(* Logix 5000 project; controller cow Emulate 5570 rev 36.11; software revision 36.00; part 2 of 6 *)

ADD_ON_INSTRUCTION RTOS_Format   (* revision 1.0 *)
VAR_INPUT
   Source : REAL; {required}
END_VAR
VAR_IN_OUT
   Dest : String20; {required}
END_VAR
VAR
   DotS : STRING := '.'; {access None}
   dotPos : DINT[2]; {access None}
   dotPos_1 : DINT; {access None}
   Blank : STRING := ' '; {access None}
END_VAR

ROUTINE Logic   (* ladder *)
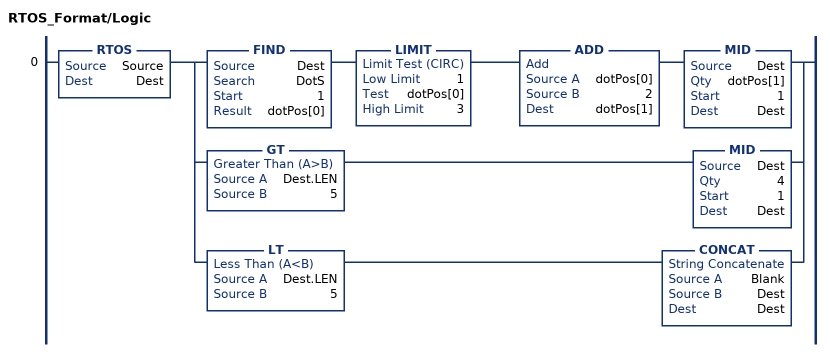
   0: RTOS(Source,Dest)[FIND(Dest,DotS,1,dotPos[0]) LIMIT(1,dotPos[0],3) ADD(dotPos[0],2,dotPos[1]) MID(Dest,dotPos[1],1,Dest) ,GT(Dest.LEN,5) MID(Dest,4,1,Dest) ,LT(Dest.LEN,5) CONCAT(Blank,Dest,Dest) ];
END_ROUTINE
END_ADD_ON_INSTRUCTION

ADD_ON_INSTRUCTION SCALE_WEIGHT   (* revision 1.0 *)
VAR_INPUT
   BCD0 : ALIAS FOR BCD.0; {access None, visible}
   BCD1 : ALIAS FOR BCD.1; {access None, visible}
   BCD2 : ALIAS FOR BCD.2; {access None, visible}
   BCD3 : ALIAS FOR BCD.3; {access None, visible}
   BCD4 : ALIAS FOR BCD.4; {access None, visible}
   BCD5 : ALIAS FOR BCD.5; {access None, visible}
   BCD6 : ALIAS FOR BCD.6; {access None, visible}
   BCD7 : ALIAS FOR BCD.7; {access None, visible}
   BCD8 : ALIAS FOR BCD.8; {access None, visible}
   BCD9 : ALIAS FOR BCD.9; {access None, visible}
   BCD10 : ALIAS FOR BCD.10; {access None, visible}
   BCD11 : ALIAS FOR BCD.11; {access None, visible}
   BCD12 : ALIAS FOR BCD.12; {access None, visible}
   BCD13 : ALIAS FOR BCD.13; {access None, visible}
   BCD14 : ALIAS FOR BCD.14; {access None, visible}
   BCD15 : ALIAS FOR BCD.15; {access None, visible}
END_VAR
VAR_OUTPUT
   DM : BOOL; {access Read Only, visible}
   DMGL : BOOL; {access Read Only, visible}
END_VAR
VAR_INPUT
   PB : BOOL; {visible}
END_VAR
VAR_OUTPUT
   SV : BOOL; {access Read Only, visible}
END_VAR
VAR_INPUT
   LL : BOOL; {visible}
END_VAR
VAR_OUTPUT
   PB2 : BOOL;
   DM2 : BOOL;
END_VAR
VAR_INPUT
   Sign : BOOL;
END_VAR
VAR_OUTPUT
   Value : INT; {access Read Only, visible}
END_VAR
VAR_IN_OUT
   Sys : Sys_Data; {required}
END_VAR
VAR
   BCD : INT; {access None}
END_VAR

ROUTINE Logic   (* ladder *)
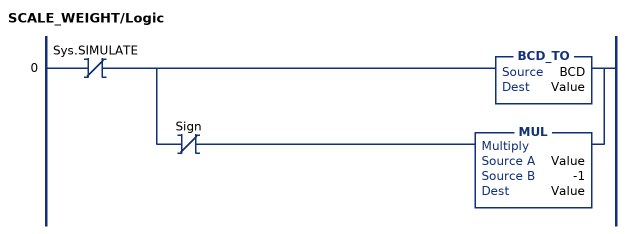
   0: XIO(Sys.SIMULATE)[BCD_TO(BCD,Value) ,XIO(Sign) MUL(Value,-1,Value) ];
END_ROUTINE
END_ADD_ON_INSTRUCTION

ADD_ON_INSTRUCTION Speed_RPM   (* revision 1.0 *)
VAR_IN_OUT
   Motor : MotorX; {required}
END_VAR
VAR_INPUT
   RPM_Low : INT := 60; {visible}
END_VAR
VAR_OUTPUT
   RPM : INT; {visible}
END_VAR
VAR
   Timer : TIMER := (PRE := 5000); {access None}
   temp : INT[10]; {access None}
   Sort_control : CONTROL := (LEN := 10); {access None}
   RPM_AVG : REAL; {access None}
   rpm_ons : DINT; {access None}
   No_Input : BOOL; {access None}
   FIFO_control : CONTROL := (LEN := 10, POS := 10); {access None}
   FIFO : INT[11]; {access None}
   AVE_Control : CONTROL := (LEN := 8); {access None}
   Motor_Start : TIMER := (PRE := 5000); {access None}
   Delay : TIMER := (PRE := 5000); {access None}
   RUNTIME : TIMER := (PRE := 14400000, ACC := 14400000); {access None}
END_VAR

ROUTINE Logic   (* ladder *)
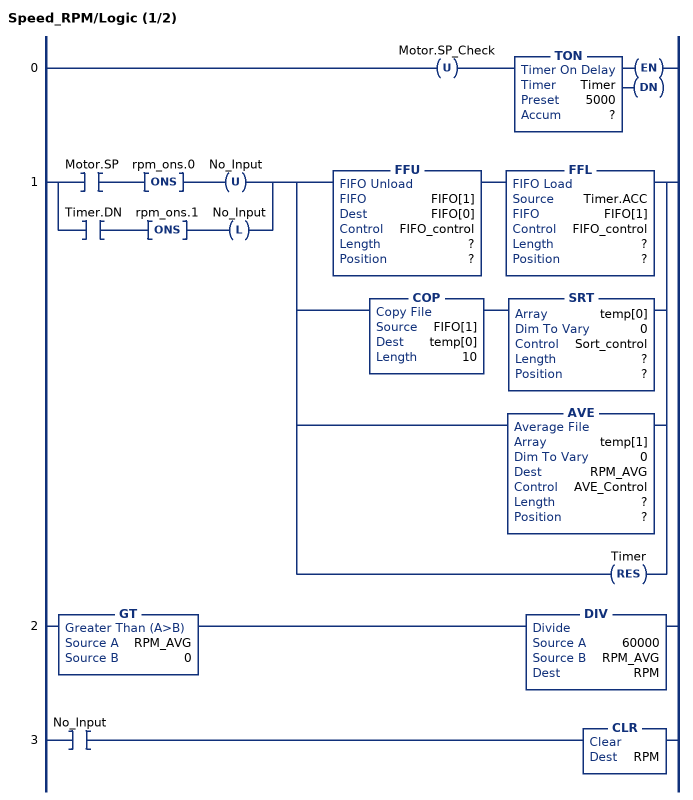
   0: OTU(Motor.SP_Check)TON(Timer,?,?);
   1: [XIC(Motor.SP) ONS(rpm_ons.0) OTU(No_Input) ,XIC(Timer.DN) ONS(rpm_ons.1) OTL(No_Input) ][FFU(FIFO[1],FIFO[0],FIFO_control,?,?) FFL(Timer.ACC,FIFO[1],FIFO_control,?,?) ,COP(FIFO[1],temp[0],10) SRT(temp[0],0,Sort_control,?,?) ,AVE(temp[1],0,RPM_AVG,AVE_Control,?,?) ,RES(Timer) ];
   2: GT(RPM_AVG,0)DIV(60000,RPM_AVG,RPM);
   3: XIC(No_Input)CLR(RPM);
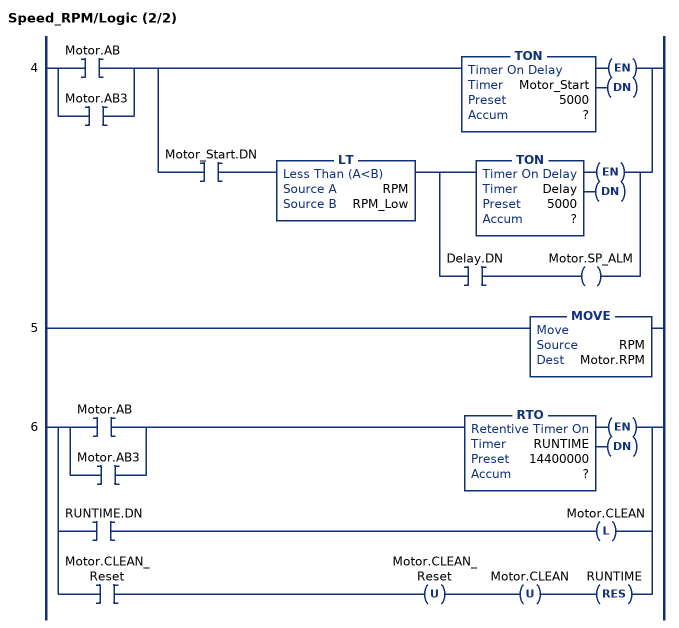
   4: [XIC(Motor.AB) ,XIC(Motor.AB3) ][TON(Motor_Start,?,?) ,XIC(Motor_Start.DN) LT(RPM,RPM_Low) [TON(Delay,?,?) ,XIC(Delay.DN) OTE(Motor.SP_ALM) ] ];
   5: MOVE(RPM,Motor.RPM);
   6: [[XIC(Motor.AB) ,XIC(Motor.AB3) ] RTO(RUNTIME,?,?) ,XIC(RUNTIME.DN) OTL(Motor.CLEAN) ,XIC(Motor.CLEAN_Reset) OTU(Motor.CLEAN_Reset) OTU(Motor.CLEAN) RES(RUNTIME) ];
END_ROUTINE
END_ADD_ON_INSTRUCTION

ADD_ON_INSTRUCTION Str_Len_Fix   (* revision 1.0 *)
VAR_IN_OUT
   Str : STRING; {required}
END_VAR
VAR_INPUT
   Len : DINT; {required}
END_VAR

ROUTINE Logic   (* ladder *)
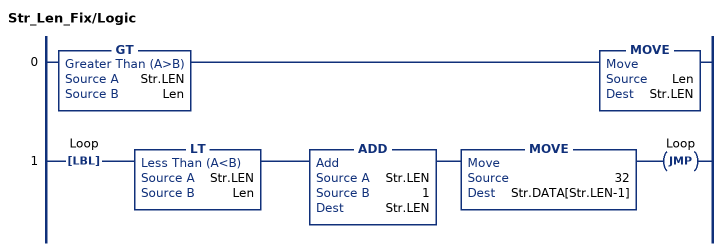
   0: GT(Str.LEN,Len)MOVE(Len,Str.LEN);
   1: LBL(Loop)LT(Str.LEN,Len)ADD(Str.LEN,1,Str.LEN)MOVE(32,Str.DATA[Str.LEN-1])JMP(Loop);
END_ROUTINE
END_ADD_ON_INSTRUCTION

ADD_ON_INSTRUCTION System_Data   (* revision 1.0 *)
VAR_OUTPUT
   MC : BOOL; {visible}
END_VAR
VAR_IN_OUT
   SYS : Sys_Data; {required}
   STS : INT; {required}
   sys_common : System_Common; {required}
END_VAR
VAR
   ons : DINT; {access None}
   EM_TIMER : TIMER := (PRE := 5000); {access None}
   BIN_SEL_PRE : DINT; {access None}
   BIN_SELS_PRE : DINT; {access None}
   Report_Log : TIMER := (PRE := 5000); {access None}
   Err_Reset_Timer : TIMER := (PRE := 1000); {access None}
END_VAR

ROUTINE Logic   (* ladder *)
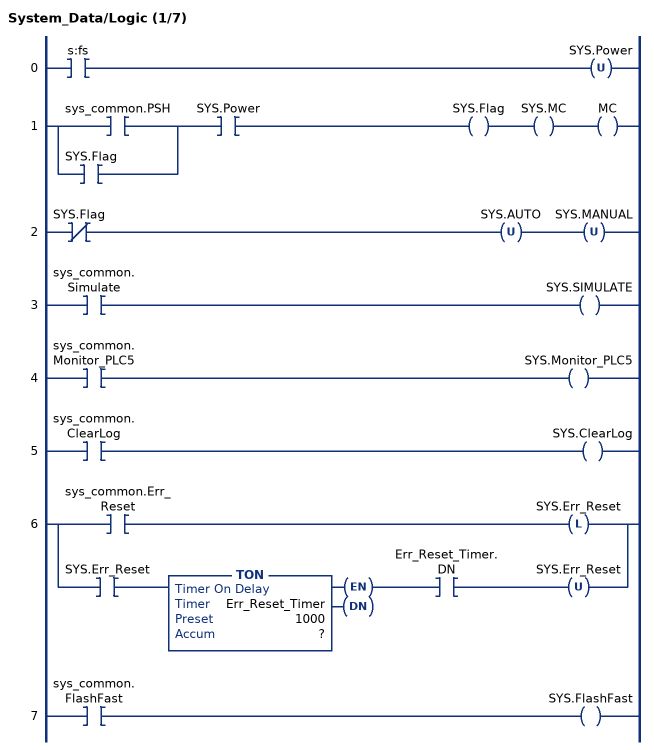
   0: XIC(s:fs)OTU(SYS.Power);
   1: [XIC(sys_common.PSH) ,XIC(SYS.Flag) ]XIC(SYS.Power)OTE(SYS.Flag)OTE(SYS.MC)OTE(MC);
   2: XIO(SYS.Flag)OTU(SYS.AUTO)OTU(SYS.MANUAL);
   3: XIC(sys_common.Simulate)OTE(SYS.SIMULATE);
   4: XIC(sys_common.Monitor_PLC5)OTE(SYS.Monitor_PLC5);
   5: XIC(sys_common.ClearLog)OTE(SYS.ClearLog);
   6: [XIC(sys_common.Err_Reset) OTL(SYS.Err_Reset) ,XIC(SYS.Err_Reset) TON(Err_Reset_Timer,?,?) XIC(Err_Reset_Timer.DN) OTU(SYS.Err_Reset) ];
   7: XIC(sys_common.FlashFast)OTE(SYS.FlashFast);
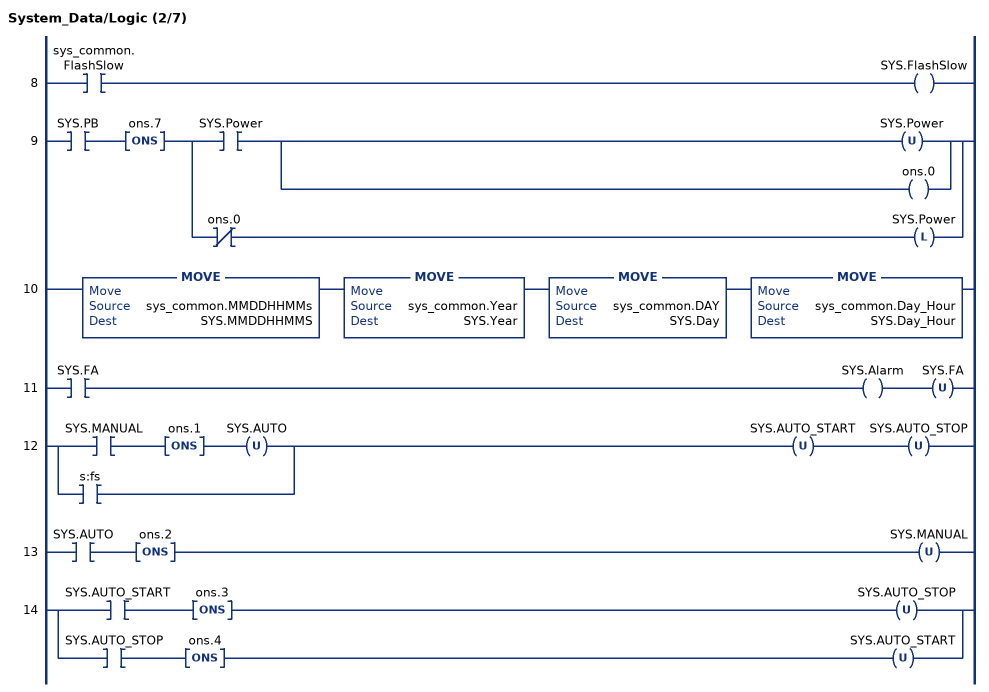
   8: XIC(sys_common.FlashSlow)OTE(SYS.FlashSlow);
   9: XIC(SYS.PB)ONS(ons.7)[XIC(SYS.Power) [OTU(SYS.Power) ,OTE(ons.0) ] ,XIO(ons.0) OTL(SYS.Power) ];
   10: MOVE(sys_common.MMDDHHMMs,SYS.MMDDHHMMS)MOVE(sys_common.Year,SYS.Year)MOVE(sys_common.DAY,SYS.Day)MOVE(sys_common.Day_Hour,SYS.Day_Hour);
   11: XIC(SYS.FA)OTE(SYS.Alarm)OTU(SYS.FA);
   12: [XIC(SYS.MANUAL) ONS(ons.1) OTU(SYS.AUTO) ,XIC(s:fs) ]OTU(SYS.AUTO_START)OTU(SYS.AUTO_STOP);
   13: XIC(SYS.AUTO)ONS(ons.2)OTU(SYS.MANUAL);
   14: [XIC(SYS.AUTO_START) ONS(ons.3) OTU(SYS.AUTO_STOP) ,XIC(SYS.AUTO_STOP) ONS(ons.4) OTU(SYS.AUTO_START) ];
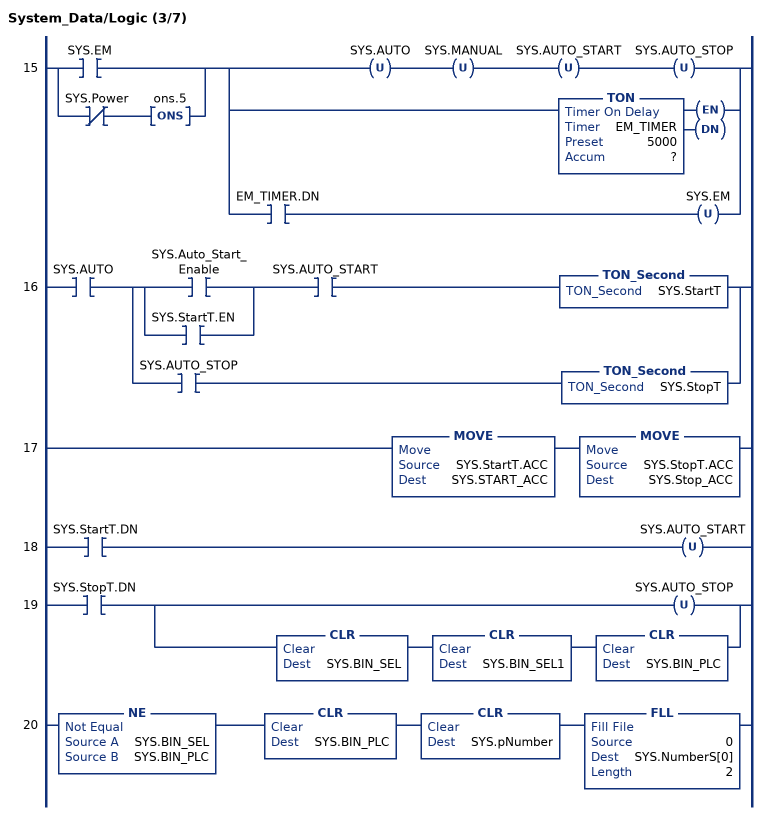
   15: [XIC(SYS.EM) ,XIO(SYS.Power) ONS(ons.5) ][OTU(SYS.AUTO) OTU(SYS.MANUAL) OTU(SYS.AUTO_START) OTU(SYS.AUTO_STOP) ,TON(EM_TIMER,?,?) ,XIC(EM_TIMER.DN) OTU(SYS.EM) ];
   16: XIC(SYS.AUTO)[[XIC(SYS.Auto_Start_Enable) ,XIC(SYS.StartT.EN) ] XIC(SYS.AUTO_START) TON_Second(SYS.StartT) ,XIC(SYS.AUTO_STOP) TON_Second(SYS.StopT) ];
   17: MOVE(SYS.StartT.ACC,SYS.START_ACC)MOVE(SYS.StopT.ACC,SYS.Stop_ACC);
   18: XIC(SYS.StartT.DN)OTU(SYS.AUTO_START);
   19: XIC(SYS.StopT.DN)[OTU(SYS.AUTO_STOP) ,CLR(SYS.BIN_SEL) CLR(SYS.BIN_SEL1) CLR(SYS.BIN_PLC) ];
   20: NE(SYS.BIN_SEL,SYS.BIN_PLC)CLR(SYS.BIN_PLC)CLR(SYS.pNumber)FLL(0,SYS.NumberS[0],2);
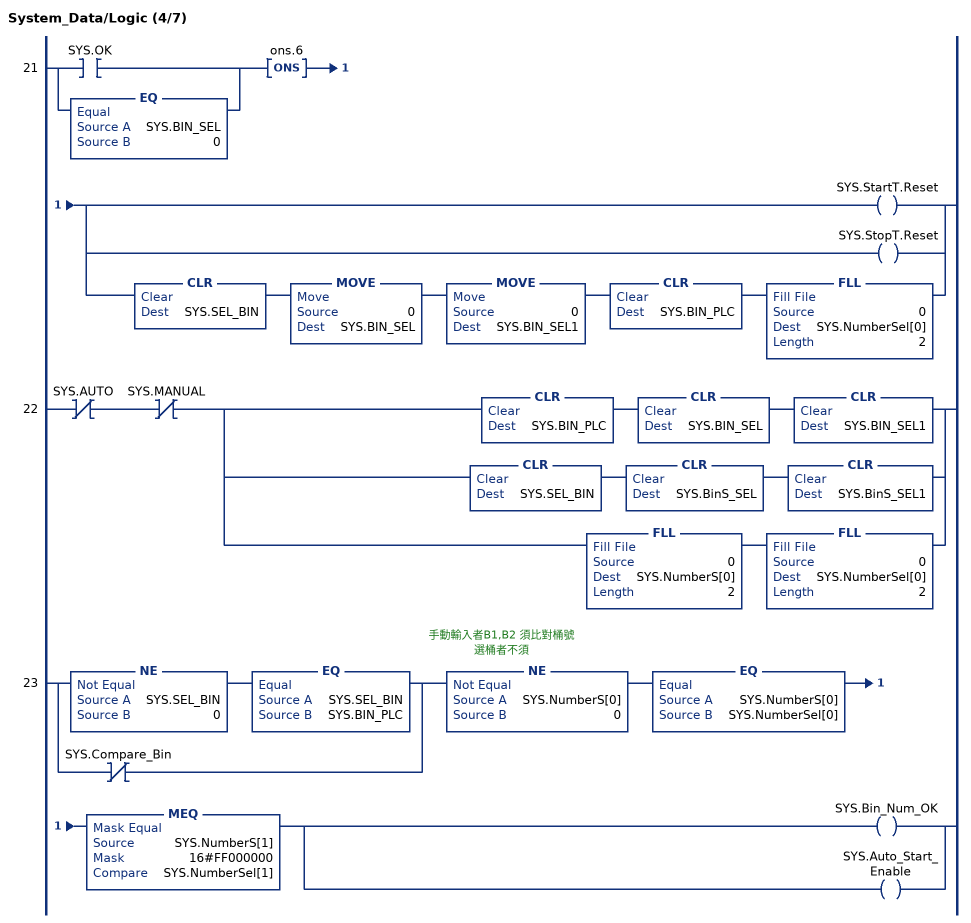
   21: [XIC(SYS.OK) ,EQ(SYS.BIN_SEL,0) ]ONS(ons.6)[OTE(SYS.StartT.Reset) ,OTE(SYS.StopT.Reset) ,CLR(SYS.SEL_BIN) MOVE(0,SYS.BIN_SEL) MOVE(0,SYS.BIN_SEL1) CLR(SYS.BIN_PLC) FLL(0,SYS.NumberSel[0],2) ];
   22: XIO(SYS.AUTO)XIO(SYS.MANUAL)[CLR(SYS.BIN_PLC) CLR(SYS.BIN_SEL) CLR(SYS.BIN_SEL1) ,CLR(SYS.SEL_BIN) CLR(SYS.BinS_SEL) CLR(SYS.BinS_SEL1) ,FLL(0,SYS.NumberS[0],2) FLL(0,SYS.NumberSel[0],2) ];
   // 手動輸入者B1,B2 須比對桶號
   // 選桶者不須
   23: [NE(SYS.SEL_BIN,0) EQ(SYS.SEL_BIN,SYS.BIN_PLC) ,XIO(SYS.Compare_Bin) ]NE(SYS.NumberS[0],0)EQ(SYS.NumberS[0],SYS.NumberSel[0])MEQ(SYS.NumberS[1],16#FF000000,SYS.NumberSel[1])[OTE(SYS.Bin_Num_OK) ,OTE(SYS.Auto_Start_Enable) ];
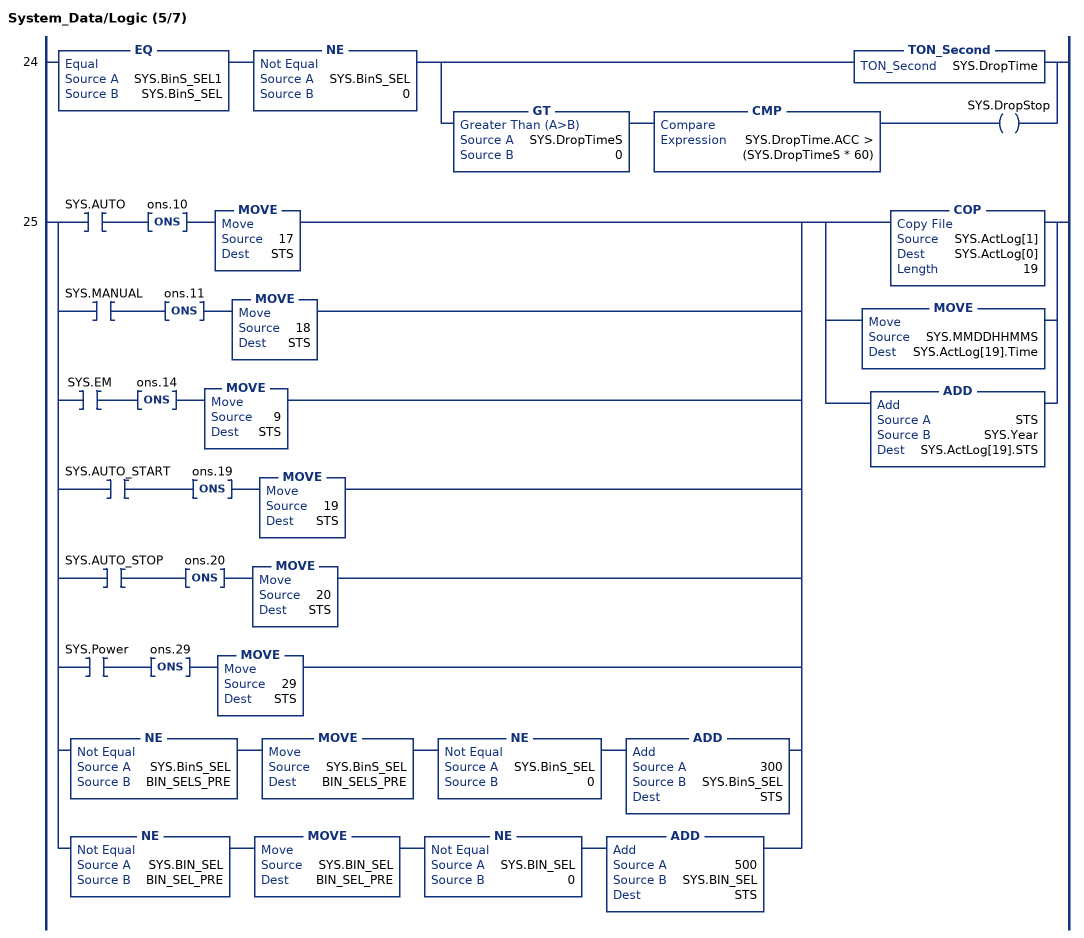
   24: EQ(SYS.BinS_SEL1,SYS.BinS_SEL)NE(SYS.BinS_SEL,0)[TON_Second(SYS.DropTime) ,GT(SYS.DropTimeS,0) CMP(SYS.DropTime.ACC > (SYS.DropTimeS * 60)) OTE(SYS.DropStop) ];
   25: [XIC(SYS.AUTO) ONS(ons.10) MOVE(17,STS) ,XIC(SYS.MANUAL) ONS(ons.11) MOVE(18,STS) ,XIC(SYS.EM) ONS(ons.14) MOVE(9,STS) ,XIC(SYS.AUTO_START) ONS(ons.19) MOVE(19,STS) ,XIC(SYS.AUTO_STOP) ONS(ons.20) MOVE(20,STS) ,XIC(SYS.Power) ONS(ons.29) MOVE(29,STS) ,NE(SYS.BinS_SEL,BIN_SELS_PRE) MOVE(SYS.BinS_SEL,BIN_SELS_PRE) NE(SYS.BinS_SEL,0) ADD(300,SYS.BinS_SEL,STS) ,NE(SYS.BIN_SEL,BIN_SEL_PRE) MOVE(SYS.BIN_SEL,BIN_SEL_PRE) NE(SYS.BIN_SEL,0) ADD(500,SYS.BIN_SEL,STS) ][COP(SYS.ActLog[1],SYS.ActLog[0],19) ,MOVE(SYS.MMDDHHMMS,SYS.ActLog[19].Time) ,ADD(STS,SYS.Year,SYS.ActLog[19].STS) ];
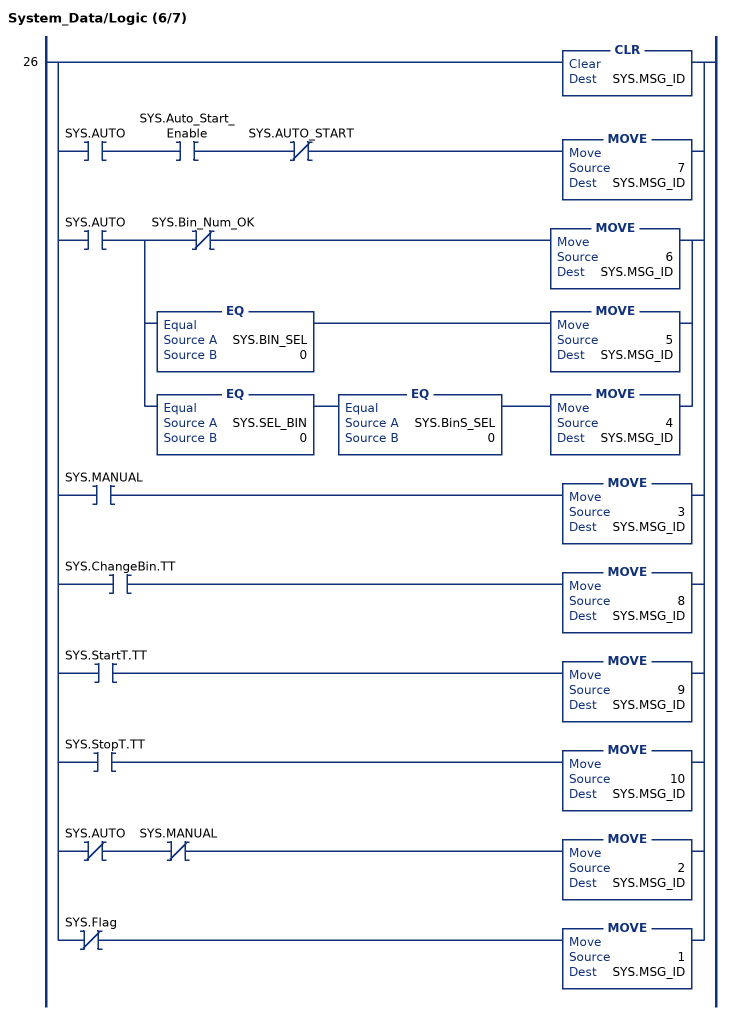
   26: [CLR(SYS.MSG_ID) ,XIC(SYS.AUTO) XIC(SYS.Auto_Start_Enable) XIO(SYS.AUTO_START) MOVE(7,SYS.MSG_ID) ,XIC(SYS.AUTO) [XIO(SYS.Bin_Num_OK) MOVE(6,SYS.MSG_ID) ,EQ(SYS.BIN_SEL,0) MOVE(5,SYS.MSG_ID) ,EQ(SYS.SEL_BIN,0) EQ(SYS.BinS_SEL,0) MOVE(4,SYS.MSG_ID) ] ,XIC(SYS.MANUAL) MOVE(3,SYS.MSG_ID) ,XIC(SYS.ChangeBin.TT) MOVE(8,SYS.MSG_ID) ,XIC(SYS.StartT.TT) MOVE(9,SYS.MSG_ID) ,XIC(SYS.StopT.TT) MOVE(10,SYS.MSG_ID) ,XIO(SYS.AUTO) XIO(SYS.MANUAL) MOVE(2,SYS.MSG_ID) ,XIO(SYS.Flag) MOVE(1,SYS.MSG_ID) ];
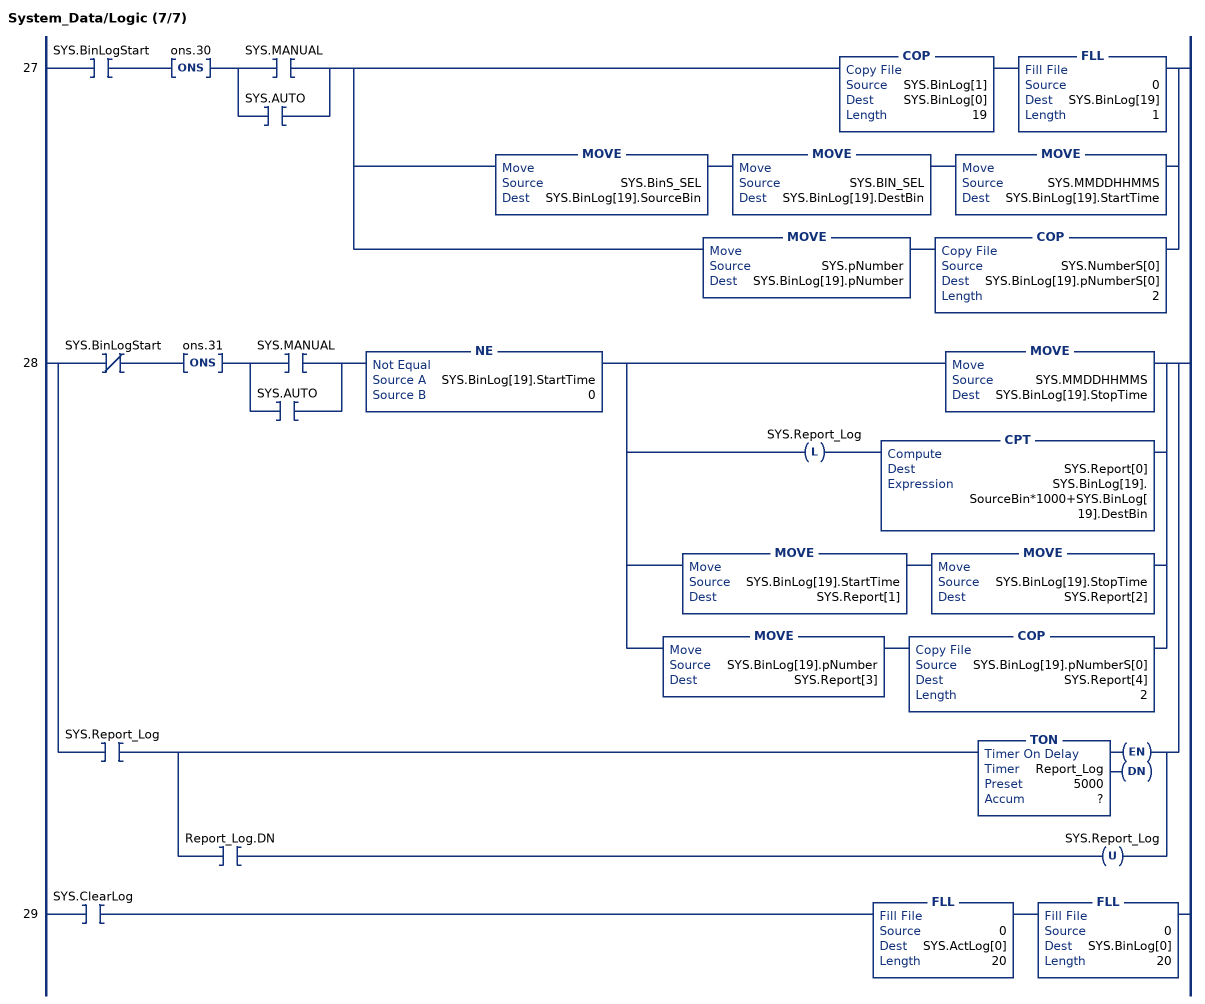
   27: XIC(SYS.BinLogStart)ONS(ons.30)[XIC(SYS.MANUAL) ,XIC(SYS.AUTO) ][COP(SYS.BinLog[1],SYS.BinLog[0],19) FLL(0,SYS.BinLog[19],1) ,MOVE(SYS.BinS_SEL,SYS.BinLog[19].SourceBin) MOVE(SYS.BIN_SEL,SYS.BinLog[19].DestBin) MOVE(SYS.MMDDHHMMS,SYS.BinLog[19].StartTime) ,MOVE(SYS.pNumber,SYS.BinLog[19].pNumber) COP(SYS.NumberS[0],SYS.BinLog[19].pNumberS[0],2) ];
   28: [XIO(SYS.BinLogStart) ONS(ons.31) [XIC(SYS.MANUAL) ,XIC(SYS.AUTO) ] NE(SYS.BinLog[19].StartTime,0) [MOVE(SYS.MMDDHHMMS,SYS.BinLog[19].StopTime) ,OTL(SYS.Report_Log) CPT(SYS.Report[0],SYS.BinLog[19].SourceBin*1000+SYS.BinLog[19].DestBin) ,MOVE(SYS.BinLog[19].StartTime,SYS.Report[1]) MOVE(SYS.BinLog[19].StopTime,SYS.Report[2]) ,MOVE(SYS.BinLog[19].pNumber,SYS.Report[3]) COP(SYS.BinLog[19].pNumberS[0],SYS.Report[4],2) ] ,XIC(SYS.Report_Log) [TON(Report_Log,?,?) ,XIC(Report_Log.DN) OTU(SYS.Report_Log) ] ];
   29: XIC(SYS.ClearLog)FLL(0,SYS.ActLog[0],20)FLL(0,SYS.BinLog[0],20);
END_ROUTINE
END_ADD_ON_INSTRUCTION

ADD_ON_INSTRUCTION TON_Second   (* revision 1.0, ExecuteEnableInFalse *)
VAR_OUTPUT
   EN : ALIAS FOR Timer.EN; {access None, visible}
   DN : ALIAS FOR Timer.DN; {access None, visible}
   TT : ALIAS FOR Timer.TT; {access None, visible}
   Reset : BOOL;
END_VAR
VAR_INPUT
   PRE : DINT; {visible}
END_VAR
VAR_OUTPUT
   ACC : DINT; {visible}
END_VAR
VAR
   Timer : TIMER; {access None}
   ACC_Temp : DINT; {access None}
END_VAR

ROUTINE EnableInFalse   (* ladder *)
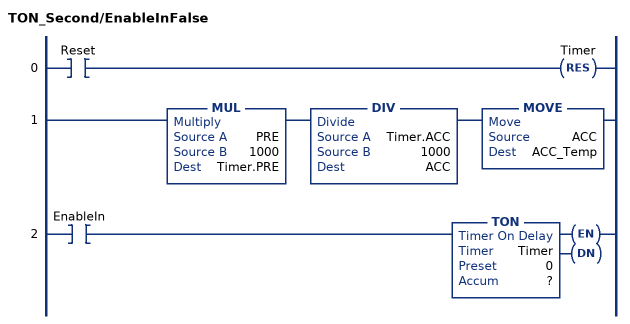
   0: XIC(Reset)RES(Timer);
   1: MUL(PRE,1000,Timer.PRE)DIV(Timer.ACC,1000,ACC)MOVE(ACC,ACC_Temp);
   2: XIC(EnableIn)TON(Timer,?,?);
END_ROUTINE

ROUTINE Logic   (* ladder *)
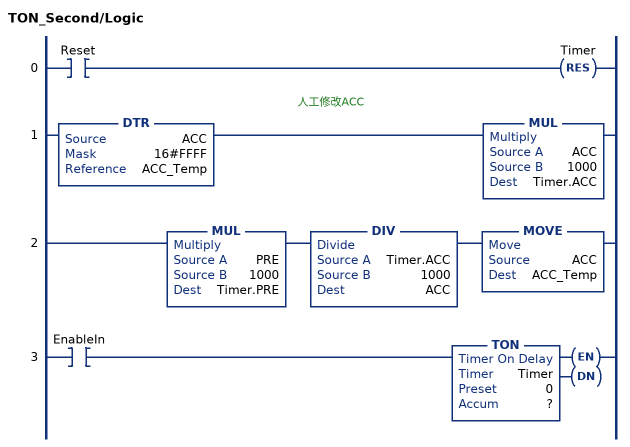
   0: XIC(Reset)RES(Timer);
   // 人工修改ACC
   1: DTR(ACC,16#FFFF,ACC_Temp)MUL(ACC,1000,Timer.ACC);
   2: MUL(PRE,1000,Timer.PRE)DIV(Timer.ACC,1000,ACC)MOVE(ACC,ACC_Temp);
   3: XIC(EnableIn)TON(Timer,?,?);
END_ROUTINE
END_ADD_ON_INSTRUCTION

ADD_ON_INSTRUCTION Valve   (* revision 1.0 *)
VAR_INPUT
   LSO : BOOL; {visible}
   LSK : BOOL; {visible}
END_VAR
VAR_OUTPUT
   SV : BOOL; {visible}
   Auto_On : BOOL;
   Manual_On : BOOL;
   Manual : BOOL; {visible}
   FA : BOOL; {visible}
   OPEN : BOOL; {visible}
   InterLock : BOOL; {access Read Only, visible}
   Auto : BOOL;
   PB : BOOL;
   GL : BOOL; {access Read Only, visible}
END_VAR
VAR_INPUT
   LL : BOOL;
END_VAR
VAR_OUTPUT
   Not_AOI_Control : BOOL; {visible}
   Lock : BOOL;
   No_Feedback : BOOL; {visible}
END_VAR
VAR_IN_OUT
   STS : INT; {required}
   Sys : Sys_Data; {required}
END_VAR
VAR
   Open_Delay : TIMER := (PRE := 500); {access None}
   Close_Delay : TIMER := (PRE := 500); {access None}
   TimeOut : TIMER := (PRE := 3000); {access None}
   Interlock_Delay : TIMER := (PRE := 500); {access None}
   ActLog : ActLog[20];
   ONS : DINT; {access None}
   LSO_Delay : TIMER := (PRE := 500); {access None}
   PB_Delay : TIMER := (PRE := 500); {access None}
   LastOnTime : DINT;
   LastOffTime : DINT;
END_VAR

ROUTINE Logic   (* ladder *)
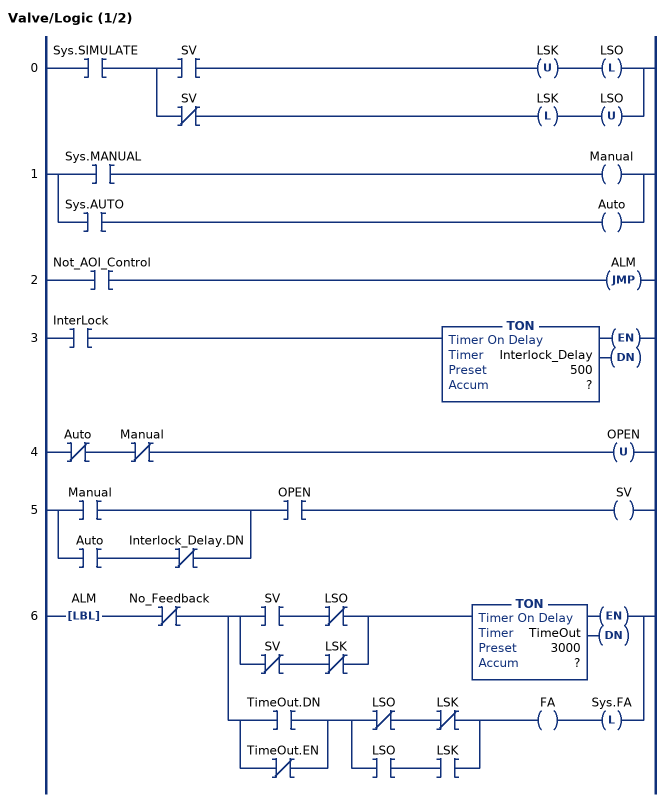
   0: XIC(Sys.SIMULATE)[XIC(SV) OTU(LSK) OTL(LSO) ,XIO(SV) OTL(LSK) OTU(LSO) ];
   1: [XIC(Sys.MANUAL) OTE(Manual) ,XIC(Sys.AUTO) OTE(Auto) ];
   2: XIC(Not_AOI_Control)JMP(ALM);
   3: XIC(InterLock)TON(Interlock_Delay,?,?);
   4: XIO(Auto)XIO(Manual)OTU(OPEN);
   5: [XIC(Manual) ,XIC(Auto) XIO(Interlock_Delay.DN) ]XIC(OPEN)OTE(SV);
   6: LBL(ALM)XIO(No_Feedback)[[XIC(SV) XIO(LSO) ,XIO(SV) XIO(LSK) ] TON(TimeOut,?,?) ,[XIC(TimeOut.DN) ,XIO(TimeOut.EN) ] [XIO(LSO) XIO(LSK) ,XIC(LSO) XIC(LSK) ] OTE(FA) OTL(Sys.FA) ];
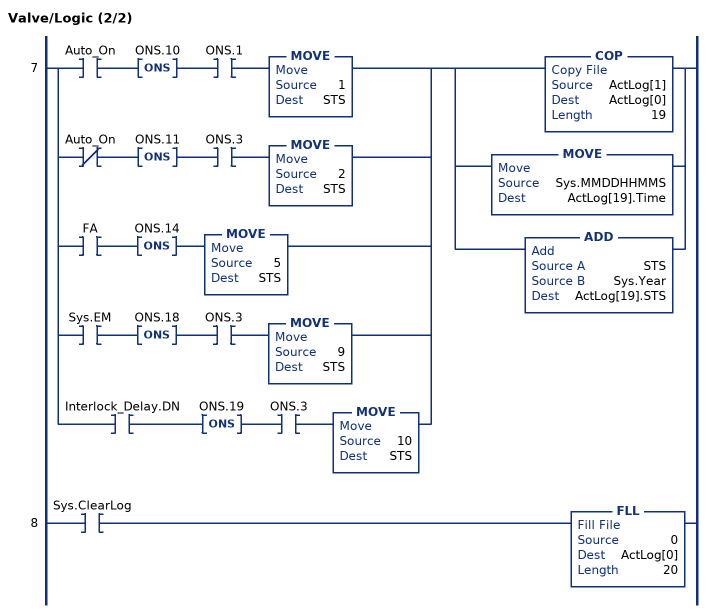
   7: [[XIC(Auto_On) ONS(ONS.10) XIC(ONS.1) MOVE(1,STS) ,XIO(Auto_On) ONS(ONS.11) XIC(ONS.3) MOVE(2,STS) ] ,XIC(FA) ONS(ONS.14) MOVE(5,STS) ,XIC(Sys.EM) ONS(ONS.18) XIC(ONS.3) MOVE(9,STS) ,XIC(Interlock_Delay.DN) ONS(ONS.19) XIC(ONS.3) MOVE(10,STS) ][COP(ActLog[1],ActLog[0],19) ,MOVE(Sys.MMDDHHMMS,ActLog[19].Time) ,ADD(STS,Sys.Year,ActLog[19].STS) ];
   8: XIC(Sys.ClearLog)FLL(0,ActLog[0],20);
END_ROUTINE
END_ADD_ON_INSTRUCTION

ADD_ON_INSTRUCTION Valve2   (* revision 1.0 *)
VAR_INPUT
   LSO : BOOL; {visible}
   LSK : BOOL; {visible}
END_VAR
VAR_OUTPUT
   SVO : BOOL; {visible}
   SVK : BOOL; {visible}
   SVOPB : BOOL;
   SVKPB : BOOL;
   Manual : BOOL; {visible}
   FA : BOOL; {visible}
   OPEN : BOOL; {visible}
   InterLock : BOOL; {access Read Only, visible}
   Auto : BOOL;
   Not_AOI_Control : BOOL; {visible}
   Lock : BOOL;
   Manual_Open : BOOL;
   Off_Delay : BOOL;
END_VAR
VAR_IN_OUT
   STS : INT; {required}
   Sys : Sys_Data; {required}
END_VAR
VAR_INPUT
   PB : BOOL;
END_VAR
VAR_OUTPUT
   GL : BOOL;
END_VAR
VAR
   TimeOut : TIMER := (PRE := 3000); {access None}
   Interlock_Delay : TIMER := (PRE := 500); {access None}
   ActLog : ActLog[20];
   ONS : DINT; {access None}
   LSO_Delay : TIMER := (PRE := 1000); {access None}
   LSK_Delay : TIMER := (PRE := 1000); {access None}
   off_delayT : TIMER := (PRE := 2000); {access None}
END_VAR

ROUTINE Logic   (* ladder *)
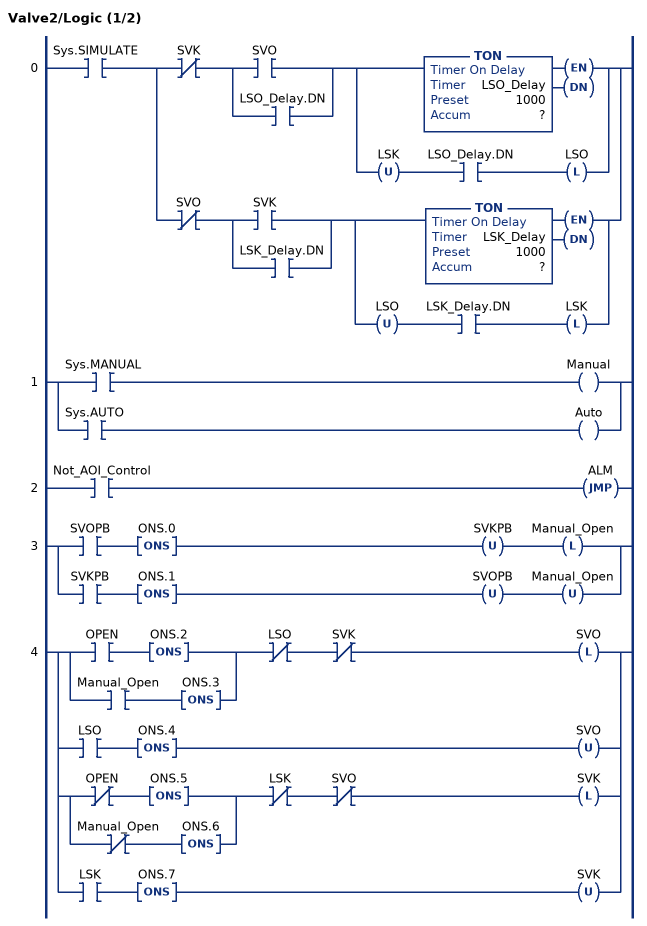
   0: XIC(Sys.SIMULATE)[XIO(SVK) [XIC(SVO) ,XIC(LSO_Delay.DN) ] [TON(LSO_Delay,?,?) ,OTU(LSK) XIC(LSO_Delay.DN) OTL(LSO) ] ,XIO(SVO) [XIC(SVK) ,XIC(LSK_Delay.DN) ] [TON(LSK_Delay,?,?) ,OTU(LSO) XIC(LSK_Delay.DN) OTL(LSK) ] ];
   1: [XIC(Sys.MANUAL) OTE(Manual) ,XIC(Sys.AUTO) OTE(Auto) ];
   2: XIC(Not_AOI_Control)JMP(ALM);
   3: [XIC(SVOPB) ONS(ONS.0) OTU(SVKPB) OTL(Manual_Open) ,XIC(SVKPB) ONS(ONS.1) OTU(SVOPB) OTU(Manual_Open) ];
   4: [[[XIC(OPEN) ONS(ONS.2) ,XIC(Manual_Open) ONS(ONS.3) ] XIO(LSO) XIO(SVK) OTL(SVO) ,XIC(LSO) ONS(ONS.4) OTU(SVO) ] ,[[XIO(OPEN) ONS(ONS.5) ,XIO(Manual_Open) ONS(ONS.6) ] XIO(LSK) XIO(SVO) OTL(SVK) ,XIC(LSK) ONS(ONS.7) OTU(SVK) ] ];
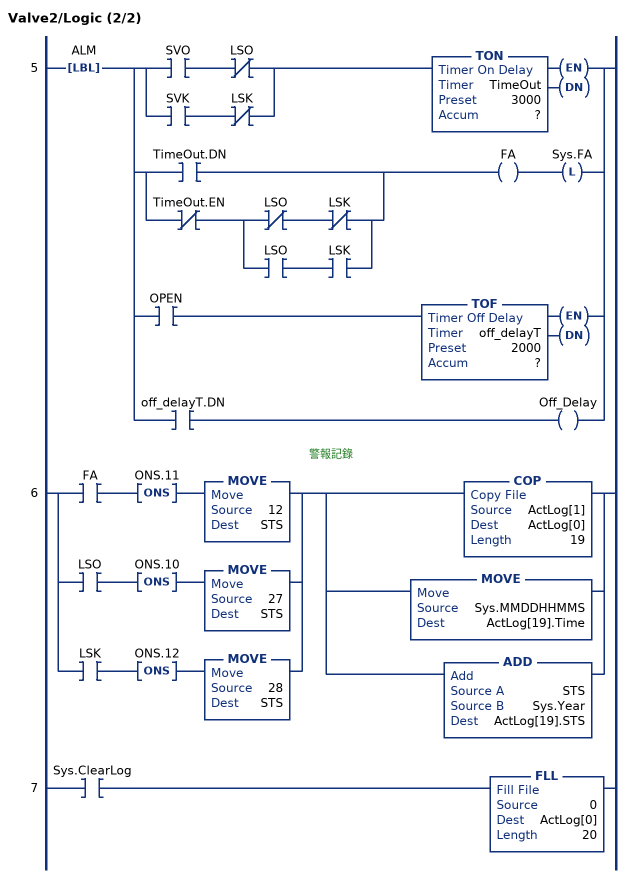
   5: LBL(ALM)[[XIC(SVO) XIO(LSO) ,XIC(SVK) XIO(LSK) ] TON(TimeOut,?,?) ,[XIC(TimeOut.DN) ,XIO(TimeOut.EN) [XIO(LSO) XIO(LSK) ,XIC(LSO) XIC(LSK) ] ] OTE(FA) OTL(Sys.FA) ,XIC(OPEN) TOF(off_delayT,?,?) ,XIC(off_delayT.DN) OTE(Off_Delay) ];
   // 警報記錄
   6: [XIC(FA) ONS(ONS.11) MOVE(12,STS) ,[XIC(LSO) ONS(ONS.10) MOVE(27,STS) ,XIC(LSK) ONS(ONS.12) MOVE(28,STS) ] ][COP(ActLog[1],ActLog[0],19) ,MOVE(Sys.MMDDHHMMS,ActLog[19].Time) ,ADD(STS,Sys.Year,ActLog[19].STS) ];
   7: XIC(Sys.ClearLog)FLL(0,ActLog[0],20);
END_ROUTINE
END_ADD_ON_INSTRUCTION
